# EPICS IOC start-up script: iocBoot/ioctec1122/meer.iocsh
drvAsynSerialPortConfigure("MEER0", "/dev/ttyUSB0", 0, 0, 0)
iocshLoad("$(IP)/iocsh/setSerialParams.iocsh","P=$(PREFIX),PORT=MEER0,BAUD=57600")
dbLoadRecords("$(ASYN)/db/asynRecord.db","P=lab:,R=asyn:meer,PORT=MEER0,ADDR=0,OMAX=0,IMAX=0")
asynOctetSetInputEos(MEER0, 0, "\r")
asynOctetSetOutputEos(MEER0, 0, "\r")
asynSetTraceIOMask(MEER0, 0, 0X1)
asynSetTraceMask(MEER0, 0, 0X1)
dbLoadRecords("$(TOP)/labApp/Db/meer.db","P=lab:meer:,ADDR=02,PORT=MEER0,SCAN=8,ASYNRECORD=lab:asyn:meer")
doAfterIocInit('dbpf("lab:meer:ChangeSpeedSEQ.PROC", "1")')
